// TIA Portal V15.1 export
// export: Created 2020-06-12T07:35:47.1943359Z, ExportSetting None, DisplayName Totally Integrated Automation Portal, DisplayVersion V15.1, DisplayName TIA Portal Openness, DisplayVersion V15.1, DisplayName STEP 7 Professional, DisplayVersion V15.1, DisplayName STEP 7 Safety, DisplayVersion V15.1, DisplayName WinCC Advanced, DisplayVersion V15.1
FUNCTION "Gas_call" : Void   // FC1000, FBD
TITLE = Gas call
{ S7_Optimized_Access := 'TRUE' }
// stored: SetENOAutomatically False
BEGIN

REGION Network 1: Control
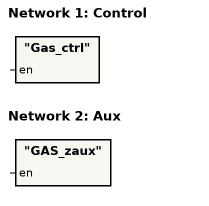
   "Gas_ctrl"();
END_REGION

REGION Network 2: Aux
   "GAS_zaux"();
END_REGION
END_FUNCTION
